ABB RAPID module: 010_conical_helix.mod

MODULE ConicalHelix
! Exercise 10 - Track a Conical Helix with the Robot
! 3D tapered spiral: Helix with linearly varying radius (e.g., widening/narrowing for conical cladding)

CONST num pi :=3.14159;                  !Pi constant
PERS num startRadius := 50;              !Initial radius (mm; taper from this)
PERS num endRadius := 100;               !Final radius (mm; > start for outward taper)
PERS num centerX := 300;                 ! Center X (base frame)
PERS num centerY := 0;                   ! Center Y (base frame)
PERS num startZ := 100;                  ! Starting Z height
PERS num pitch := 20;                    ! Z rise per turn (mm/turn)
PERS num numTurns := 9;                  ! Numbers of revolutions
PERS num segmentsPerTurn := 36;          ! Segments per revolution
PERS robtarget pHome := [[400, 0, 500], [1,0,0,0], [0,0,0,0], [9E9,9E9,9E9,9E9,9E9,9E9]];  ! Safe home

PROC main()
  VAR num totalSegments;                 ! turns * segmentsPerTurn
  VAR num angleStep;                     ! Delta theta/segment (rad)
  VAR num currentAngle := 0;             ! Cumulative angle
  VAR num currentZ := startZ;            ! Progressive Z
  VAR num currentRadius := startradius;  ! Interpolated radius
  VAR num radiusStep;                    ! Delta radius per segment
  VAR robtarget pCurrent;                ! Current pose
  VAR robtarget pNext;                   ! Next pose

  ! Derive params: radiusStep = (end - start) / totalSegments for linear taper
  totalSegments := numTurns * segmentsPerTurn;
  angleStep := 2 * pi/segmentsPerTurn;
  radiusStep := (endRadius - startRadius)/totalSegments;    ! Positive for outward, negative for inward

  ! Approach home
  MoveJ pHome, v500, z50, tool0;

  ! Start point: θ=0, r=startRadius, Z=startZ
  pCurrent := [[centerX + startRadius * Cos(0), centerY + startRadius * Sin(0), startZ],[1,0,0,0], [0,0,0,0], [9E9,9E9,9E9,9E9,9E9,9E9]];
  MoveL pCurrent, v200, fine, tool0;

  ! Conical helix loop: Update r, θ, Z per segment
  FOR i FROM 1 TO totalSegments DO
    currentAngle := currentAngle + angleStep;    ! Cumulative

    ! Radius interpolation: Linear change = start + i * step
    currentRadius := startRadius + i * radiusStep;

    ! Z interpolation: As before, fractional * total height
    currentZ := startZ + (i/totalSegments) * (pitch * numTurns);

    ! Parametric pose: Variable r in Cos/Sin
    pNext := [[centerX + currentRadius * Cos(currentAngle),
          centerY + currentRadius * Sin(currentAngle),
          currentZ],
          [1,0,0,0}, [0,0,0,0], [9E9,9E9,9E9,9E9,9E9,9E9]];

    MoveL pNext, v100, z1, tool0;  ! Segment move

    pCurrent := pNext;
  ENDFOR

  ! Retract home
  MoveJ pHome, v500, z50, tool0;
  TPWrite "Conical helix complete: Taper from " \Num:=startRadius \ "to "\Num:=endRadius \ " mm";
ENDPROC

ENDMODULE
